// EtherCatMaster with its hardware inputs and slave arrays fed from the test instead of the master
// device. Exposes the protected evaluation steps so they can be driven without ADS or an EtherCAT master.
FUNCTION_BLOCK EtherCatMaster_Mockup EXTENDS EtherCatMaster<1, 1>
VAR
END_VAR

// Same inputs as EtherCatMaster.FB_Init; the base constructor receives them implicitly.
METHOD FB_Init : BOOL
VAR_INPUT
	bInitRetains	: BOOL; // TRUE: the retain variables are initialized (reset warm / reset cold)
	bInCopyCode		: BOOL; // TRUE: the instance will be copied to the copy code afterward (online change)
	Name			: T_MaxString;
	EcStartupCycles : UINT;
END_VAR
END_METHOD

// Current step of the slave diagnostic sequence (0 = idle).
PROPERTY DiagnosticStep : UDINT
GET
DiagnosticStep := SlaveSequence;
END_GET
END_PROPERTY

// Fakes a finished Initialize: Count slaves named Slave1..SlaveN at addresses 1001.., all OP, no mailbox.
METHOD LoadConfiguration
VAR_INPUT
	Count : UINT;
END_VAR

VAR
	i : UINT;
	n : UINT;
END_VAR
n := MIN(Count, MAX_EC_SLAVES + 1);

EcMaster.CfgSlaveCount := n;
EcMaster.SlaveCount	   := n;
SlaveCountUsed		   := n;

i := 0;
WHILE i < n DO
	ConfiguredSlaveInfo[i].nAddr		  := FIRST_SLAVE_ADDR + i;
	ConfiguredSlaveInfo[i].sName		  := CONCAT('Slave', TO_STRING(i + 1));
	ConfiguredSlaveInfo[i].nMailboxInSize := 0;
	SlavesState[i].deviceState			  := 16#08; // OP
	SlavesState[i].linkState			  := 16#00;
	SlaveTopologyInfo[i].nStatusBits	  := 0;	// no hot connect group (see SetHotConnect)
	IoDevice[i].Name					  := ConfiguredSlaveInfo[i].sName;
	IoDevice[i].State					  REF= SlavesState[i];
	IoDevice[i].Configuration			  REF= ConfiguredSlaveInfo[i];
	i									  := i + 1;
END_WHILE

BuildAddrToIndex();
Initialized := TRUE;
END_METHOD

// One evaluation of the master DevState (normally done by CyclicLogic).
METHOD RunMasterState : BOOL
RunMasterState := MasterState();
END_METHOD

// One cycle of the slave diagnostic sequence (normally done by CyclicLogic).
METHOD RunSlaveState
SlaveState();
_Busy := SlaveSequence <> 0;
END_METHOD

// Target of the diagnostic ADS reads (normally taken from EcMaster.AmsNetID in Initialize).
METHOD SetMasterAmsNetId
VAR_INPUT
	NetId : T_AmsNetId;
END_VAR
_MasterAmsNetId := NetId;
END_METHOD

// Fakes the master process image: DevState word and number of slaves currently on the bus.
METHOD SetMasterDevState
VAR_INPUT
	DevState   : UINT;
	SlaveCount : UINT;
END_VAR
EcMaster.DevState	:= DevState;
EcMaster.SlaveCount := SlaveCount;
END_METHOD

// Gives the configured slave Index another EtherCAT address and rebuilds the address map.
METHOD SetSlaveAddress
VAR_INPUT
	Index : UINT;
	Addr  : UINT;
END_VAR
ConfiguredSlaveInfo[Index].nAddr := Addr;
BuildAddrToIndex();
END_METHOD

// Fakes the topology read: marks one slave as member of a hot connect group.
METHOD SetHotConnect
VAR_INPUT
	Index : UINT;
END_VAR
SlaveTopologyInfo[Index].nStatusBits.4 := TRUE;
END_METHOD

// Fakes the state read of one slave.
METHOD SetSlaveState
VAR_INPUT
	Index		: UINT;
	DeviceState : BYTE;
	LinkState	: BYTE;
END_VAR
SlavesState[Index].deviceState := DeviceState;
SlavesState[Index].linkState   := LinkState;
END_METHOD

// Requests a slave diagnostic sequence (normally triggered by ChangeCount, slave count or frame WC state).
METHOD StartDiagnostic
RunSlaveDiag := TRUE;
END_METHOD

END_FUNCTION_BLOCK

(* stored: Version 1.1.0.1, ProductVersion 3.1.4026.18
   POU EtherCatMaster_Mockup: Id {5d8d3455-3037-4a3a-8f07-a6cec3895f39}, SpecialFunc None
   Method FB_Init: Id {0d450fdf-169c-4d12-a5b5-3c33a2d8fce1}
   Property DiagnosticStep: Id {e5d0ea0a-5401-4c8d-8ba4-9ee1b295ed2c}
   Get Get: Id {446d9455-319b-4b82-8468-ef4cebd205f1}
   Method LoadConfiguration: Id {d3c3ed95-6243-4255-abab-edace0fc2cf2}
   Method RunMasterState: Id {1940fc6d-5d5b-4880-beef-e977459012da}
   Method RunSlaveState: Id {0ed23de3-fcaf-4de5-8c0b-d816862db89b}
   Method SetMasterAmsNetId: Id {f94dbf8f-fea0-4483-a83b-80aaaab3ba93}
   Method SetMasterDevState: Id {3b7d2612-ff38-4288-a5c9-7f10ded4bbd2}
   Method SetSlaveAddress: Id {8242f82f-a124-42c3-afca-8c5bfbbc8d5e}
   Method SetHotConnect: Id {3507781b-af48-492d-af78-5b1087afd038}
   Method SetSlaveState: Id {701d6f27-147a-4bc3-82f0-f67c51db7b15}
   Method StartDiagnostic: Id {cf46a52b-7bc4-415d-9653-5f48215c363f} *)
